PROGRAM Convert
VAR
	Timer:INT;
END_VAR

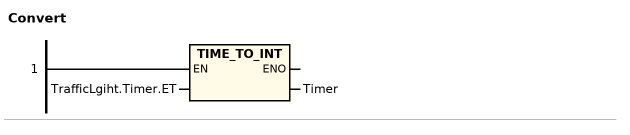
// NETWORK 1
Timer := TIME_TO_INT(TrafficLgiht.Timer.ET);

END_PROGRAM

(* stored: Version 1.1.0.1, ProductVersion 3.1.4024.11
   POU Convert: Id {0ae7e386-c154-4d31-8e31-63c23e09a0d5}, SpecialFunc None *)
